// TIA Portal project "Water Transfer and Filtration" (V17)
// Water Treatment Plant
// Start the water pump to transfer the water. Then filtration for 30 sec, then addition of chemicals for 5 sec. And then Pump 2 will be ON to transfer water into storage tank

(* hardware
DEVICE "S7-1200 station_1"  S7-1200 Station
   slot 0: "Rack_0"  S7-1200 Rack  Rack  V1.0
   slot 1: "PLC_1"  CPU 1215C DC/DC/Rly  6ES7 215-1HG40-0XB0  V4.5
*)

// ===== PLC "PLC_1"  CPU 1215C DC/DC/Rly =====

VAR_GLOBAL   // PLC tag table "Default tag table"
   "Start button P1" AT %I0.0 : Bool;
   "Start button P2" AT %I0.1 : Bool;
   "filtration" AT %Q0.0 : Bool;
   "Add chemicals" AT %Q0.1 : Bool;
   "transfer" AT %Q0.2 : Bool;
   "Pump1" AT %Q0.3 : Bool;
   "Pump2" AT %Q0.4 : Bool;
   "Tag_1" AT %M0.0 : Bool;
END_VAR

// folder: System blocks/Program resources

DATA_BLOCK "IEC_Timer_0_DB"   // DB1
{ S7_Optimized_Access := 'TRUE' }
AUTHOR : Simatic
FAMILY : IEC
NAME : IEC_TMR
VERSION : 1.0
// stored: InstanceOfName IEC_TIMER
"IEC_TIMER"
BEGIN
END_DATA_BLOCK

DATA_BLOCK "IEC_Timer_0_DB_1"   // DB2
{ S7_Optimized_Access := 'TRUE' }
AUTHOR : Simatic
FAMILY : IEC
NAME : IEC_TMR
VERSION : 1.0
// stored: InstanceOfName IEC_TIMER
"IEC_TIMER"
BEGIN
END_DATA_BLOCK

DATA_BLOCK "IEC_Timer_0_DB_2"   // DB3
{ S7_Optimized_Access := 'TRUE' }
AUTHOR : Simatic
FAMILY : IEC
NAME : IEC_TMR
VERSION : 1.0
// stored: InstanceOfName IEC_TIMER
"IEC_TIMER"
BEGIN
END_DATA_BLOCK

// folder: (top level)

ORGANIZATION_BLOCK "Main"   // OB1, LAD, ProgramCycle
TITLE = "Main Program Sweep (Cycle)"
{ S7_Optimized_Access := 'TRUE' }
VERSION : 0.1
   VAR_INPUT
      Initial_Call : Bool;   // Initial call of this OB
      Remanence : Bool;   // =True, if remanent data are available
   END_VAR
BEGIN

REGION Network 1
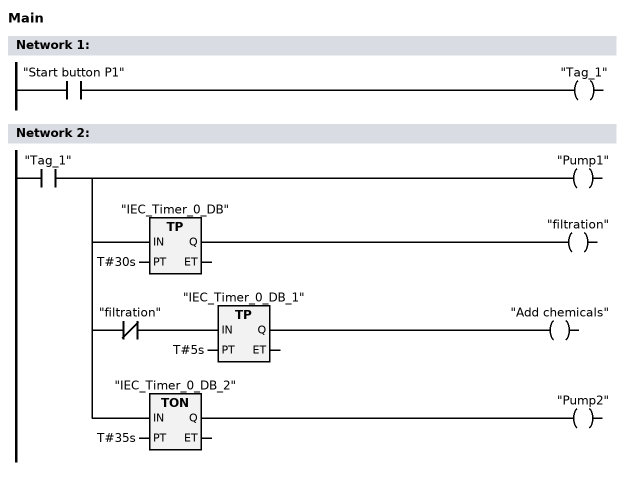
   RUNG wire#powerrail
      Contact( "Start button P1" )
      Coil( "Tag_1" )
   END_RUNG
   // the same network as SCL:
   "Tag_1" := "Start button P1";
END_REGION

REGION Network 2
   "Pump1" := "Tag_1";
   "IEC_Timer_0_DB".TP(IN := "Tag_1", PT := T#30s);
   "filtration" := "IEC_Timer_0_DB".Q;
   "IEC_Timer_0_DB_1".TP(IN := "Tag_1" AND NOT "filtration", PT := T#5s);
   "Add chemicals" := "IEC_Timer_0_DB_1".Q;
   "IEC_Timer_0_DB_2".TON(IN := "Tag_1", PT := T#35s);
   "Pump2" := "IEC_Timer_0_DB_2".Q;
END_REGION
END_ORGANIZATION_BLOCK